FUNCTION_BLOCK DateAndTimeComparer EXTENDS Object IMPLEMENTS IComparer
VAR
	_ClassName : STRING := __POUNAME();
END_VAR

{attribute 'monitoring' := 'call'}
PROPERTY ClassName : STRING
GET
ClassName := _ClassName;
END_GET
END_PROPERTY

{attribute "object_name" := "Compare"}
METHOD Compare : COMPARISION_RESULT
VAR_INPUT
	left : GENERIC_VALUE;
	right : GENERIC_VALUE;
END_VAR
VAR
	leftPointer : POINTER TO DATE_AND_TIME; 
	rightPointer : POINTER TO DATE_AND_TIME; 
END_VAR
IF left.Address = 0 AND right.Address = 0 THEN
	Compare := COMPARISION_RESULT.EQUALS;
	RETURN;
END_IF

IF left.Address = 0 THEN
	Compare := COMPARISION_RESULT.LEFT_LESS_RIGHT;
	RETURN;	
END_IF

IF right.Address = 0 THEN
	Compare := COMPARISION_RESULT.LEFT_GREATER_RIGHT;
	RETURN;	
END_IF

leftPointer := left.Address;
rightPointer := right.Address;

IF leftPointer^ < rightPointer^ THEN
	Compare := COMPARISION_RESULT.LEFT_LESS_RIGHT;
ELSIF leftPointer^ > rightPointer^ THEN
	Compare := COMPARISION_RESULT.LEFT_GREATER_RIGHT;
ELSE
	Compare := COMPARISION_RESULT.EQUALS;	
END_IF
END_METHOD

{attribute 'monitoring' := 'call'}
PROPERTY Size : ULINT
GET
Size := XSIZEOF(THIS^);
END_GET
END_PROPERTY

END_FUNCTION_BLOCK

(* stored: Version 1.1.0.1
   POU DateAndTimeComparer: Id {c7624954-7866-4335-b6ea-542bbc0f5ff3}, SpecialFunc None
   Property ClassName: Id {c7158c9a-41c2-4bf7-b154-cda0e5f6fe61}
   Get Get: Id {3cf85dee-d11d-4346-a9bd-dcb2db67323b}
   Method Compare: Id {5fa917ff-f4ed-433b-afa5-de1963f626e1}
   Property Size: Id {b6e75391-1b1f-46f9-9a33-6f5c36086d2b}
   Get Get: Id {ca34781c-13ed-4e6c-a3d9-106c7d41417a} *)
